INTERFACE I_ActuatorOnOff EXTENDS I_ActuatorBase

{attribute 'monitoring' := 'call'}
PROPERTY public isOn : BOOL
GET
END_GET
END_PROPERTY

METHOD public switchOn : BOOL
VAR_INPUT
END_VAR
END_METHOD

END_INTERFACE

(* stored: Version 1.1.0.1, ProductVersion 3.1.4024.3
   Itf I_ActuatorOnOff: Id {a8aef601-0c88-4733-9ead-ab1b0ed39c2e}
   Property isOn: Id {2c2ab8aa-eb5d-4a6b-aca6-cb4dcfad0572}
   Get Get: Id {39a518e0-fbc9-4fa3-8d62-b6c7981603a9}
   Method switchOn: Id {9d2db45b-3b4c-4b66-baf8-8a9f37ad9c0a} *)
